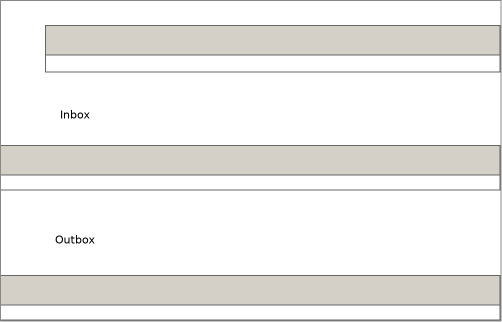
VISUALIZATION Frame_Peer  // 502x322
VAR_IN_OUT
	vio_fbPeer : FB_Peer;
	vio_stMailbox : ST_MAILBOX;
END_VAR
    Table (45,25 455x47), data array: vio_fbPeer.stMailbox
        p3854506369: vio_fbPeer.stMailbox.stInbox
        p1892666644: vio_fbPeer.stMailbox.stOutbox
        p338671338: vio_fbPeer.stMailbox.bNewMessageAvail
        p2170511999: vio_fbPeer.stMailbox.bSendingMessage
        p3723444502: vio_fbPeer.stMailbox.bMessageSent
        p1218418051: vio_fbPeer.stMailbox.eMessage
        p746581629: vio_fbPeer.stMailbox.ePeer
        p3104783080: vio_fbPeer.stMailbox.eDeliveryStatus
        p1755163831: New message avail
        p4092479075: Sending message
        p2237128397: Message sent
    Table (0,275 500x45), data array: vio_stMailbox.stOutbox
        p3854506369: vio_stMailbox.stOutbox.eMessage
        p1892666644: vio_stMailbox.stOutbox.ePeer
        p2170511999: vio_stMailbox.bSendingMessage
        p3723444502: vio_stMailbox.bMessageSent
        p338671338: vio_stMailbox.stOutbox.eDeliveryStatus
        p1755163831: Delivery Status
    Label (0,100 150x30), "Inbox"
    Label (0,225 150x30), "Outbox"
    Table (0,145 500x45), data array: vio_stMailbox.stInbox
        p3854506369: vio_stMailbox.stInbox.eMessage
        p1892666644: vio_stMailbox.stInbox.ePeer
        p2170511999: vio_stMailbox.bSendingMessage
        p3723444502: vio_stMailbox.bMessageSent
        p338671338: vio_stMailbox.stInbox.eDeliveryStatus
        p1755163831: Delivery Status
END_VISUALIZATION

(* stored: Version 1.1.0.1, ProductVersion 3.1.4024.0
   Visu Frame_Peer: Id {b3fdae91-e647-418f-93a9-e79a6fbe7143} *)
